TYPE EM_TransportCanSupply2_WRN :
STRUCT
END_STRUCT
END_TYPE

(* stored: Version 1.1.0.1, ProductVersion 3.1.4024.12
   DUT EM_TransportCanSupply2_WRN: Id {1f502c4b-2dc3-4b76-8c07-e83953e20a29} *)
